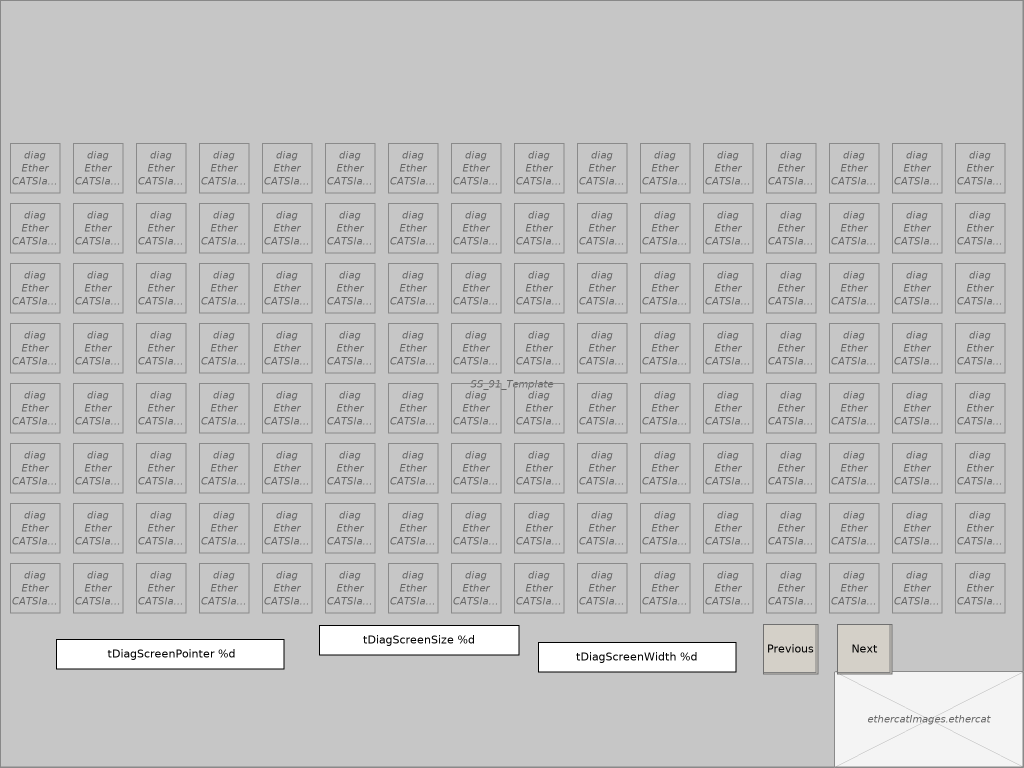
VISUALIZATION DI_02_EtherCAT  // 1024x768
    Frame (0,0 1024x768)
        shows SS_91_Template(header := HMIData.hmiHeader)
    Frame (10,143 50x50)
        shows diagEtherCATSlave(dataValues := etherCATdiag.diagScreen[1])
    Frame (73,143 50x50)
        shows diagEtherCATSlave(dataValues := etherCATdiag.diagScreen[2])
    Frame (136,143 50x50)
        shows diagEtherCATSlave(dataValues := etherCATdiag.diagScreen[3])
    Frame (199,143 50x50)
        shows diagEtherCATSlave(dataValues := etherCATdiag.diagScreen[4])
    Frame (262,143 50x50)
        shows diagEtherCATSlave(dataValues := etherCATdiag.diagScreen[5])
    Frame (325,143 50x50)
        shows diagEtherCATSlave(dataValues := etherCATdiag.diagScreen[6])
    Frame (388,143 50x50)
        shows diagEtherCATSlave(dataValues := etherCATdiag.diagScreen[7])
    Frame (451,143 50x50)
        shows diagEtherCATSlave(dataValues := etherCATdiag.diagScreen[8])
    Frame (514,143 50x50)
        shows diagEtherCATSlave(dataValues := etherCATdiag.diagScreen[9])
    Frame (577,143 50x50)
        shows diagEtherCATSlave(dataValues := etherCATdiag.diagScreen[10])
    Frame (640,143 50x50)
        shows diagEtherCATSlave(dataValues := etherCATdiag.diagScreen[11])
    Frame (703,143 50x50)
        shows diagEtherCATSlave(dataValues := etherCATdiag.diagScreen[12])
    Frame (766,143 50x50)
        shows diagEtherCATSlave(dataValues := etherCATdiag.diagScreen[13])
    Frame (829,143 50x50)
        shows diagEtherCATSlave(dataValues := etherCATdiag.diagScreen[14])
    Frame (892,143 50x50)
        shows diagEtherCATSlave(dataValues := etherCATdiag.diagScreen[15])
    Frame (955,143 50x50)
        shows diagEtherCATSlave(dataValues := etherCATdiag.diagScreen[16])
    Image (834,671 190x96), image: ethercatImages.ethercat
    Frame (10,203 50x50)
        shows diagEtherCATSlave(dataValues := etherCATdiag.diagScreen[17])
    Frame (73,203 50x50)
        shows diagEtherCATSlave(dataValues := etherCATdiag.diagScreen[18])
    Frame (136,203 50x50)
        shows diagEtherCATSlave(dataValues := etherCATdiag.diagScreen[19])
    Frame (199,203 50x50)
        shows diagEtherCATSlave(dataValues := etherCATdiag.diagScreen[20])
    Frame (262,203 50x50)
        shows diagEtherCATSlave(dataValues := etherCATdiag.diagScreen[21])
    Frame (325,203 50x50)
        shows diagEtherCATSlave(dataValues := etherCATdiag.diagScreen[22])
    Frame (388,203 50x50)
        shows diagEtherCATSlave(dataValues := etherCATdiag.diagScreen[23])
    Frame (451,203 50x50)
        shows diagEtherCATSlave(dataValues := etherCATdiag.diagScreen[24])
    Frame (514,203 50x50)
        shows diagEtherCATSlave(dataValues := etherCATdiag.diagScreen[25])
    Frame (577,203 50x50)
        shows diagEtherCATSlave(dataValues := etherCATdiag.diagScreen[26])
    Frame (640,203 50x50)
        shows diagEtherCATSlave(dataValues := etherCATdiag.diagScreen[27])
    Frame (703,203 50x50)
        shows diagEtherCATSlave(dataValues := etherCATdiag.diagScreen[28])
    Frame (766,203 50x50)
        shows diagEtherCATSlave(dataValues := etherCATdiag.diagScreen[29])
    Frame (829,203 50x50)
        shows diagEtherCATSlave(dataValues := etherCATdiag.diagScreen[30])
    Frame (892,203 50x50)
        shows diagEtherCATSlave(dataValues := etherCATdiag.diagScreen[31])
    Frame (955,203 50x50)
        shows diagEtherCATSlave(dataValues := etherCATdiag.diagScreen[32])
    Frame (10,263 50x50)
        shows diagEtherCATSlave(dataValues := etherCATdiag.diagScreen[33])
    Frame (73,263 50x50)
        shows diagEtherCATSlave(dataValues := etherCATdiag.diagScreen[34])
    Frame (136,263 50x50)
        shows diagEtherCATSlave(dataValues := etherCATdiag.diagScreen[35])
    Frame (199,263 50x50)
        shows diagEtherCATSlave(dataValues := etherCATdiag.diagScreen[36])
    Frame (262,263 50x50)
        shows diagEtherCATSlave(dataValues := etherCATdiag.diagScreen[37])
    Frame (325,263 50x50)
        shows diagEtherCATSlave(dataValues := etherCATdiag.diagScreen[38])
    Frame (388,263 50x50)
        shows diagEtherCATSlave(dataValues := etherCATdiag.diagScreen[39])
    Frame (451,263 50x50)
        shows diagEtherCATSlave(dataValues := etherCATdiag.diagScreen[40])
    Frame (514,263 50x50)
        shows diagEtherCATSlave(dataValues := etherCATdiag.diagScreen[41])
    Frame (577,263 50x50)
        shows diagEtherCATSlave(dataValues := etherCATdiag.diagScreen[42])
    Frame (640,263 50x50)
        shows diagEtherCATSlave(dataValues := etherCATdiag.diagScreen[43])
    Frame (703,263 50x50)
        shows diagEtherCATSlave(dataValues := etherCATdiag.diagScreen[44])
    Frame (766,263 50x50)
        shows diagEtherCATSlave(dataValues := etherCATdiag.diagScreen[45])
    Frame (829,263 50x50)
        shows diagEtherCATSlave(dataValues := etherCATdiag.diagScreen[46])
    Frame (892,263 50x50)
        shows diagEtherCATSlave(dataValues := etherCATdiag.diagScreen[47])
    Frame (955,263 50x50)
        shows diagEtherCATSlave(dataValues := etherCATdiag.diagScreen[48])
    Frame (10,323 50x50)
        shows diagEtherCATSlave(dataValues := etherCATdiag.diagScreen[49])
    Frame (73,323 50x50)
        shows diagEtherCATSlave(dataValues := etherCATdiag.diagScreen[50])
    Frame (136,323 50x50)
        shows diagEtherCATSlave(dataValues := etherCATdiag.diagScreen[51])
    Frame (199,323 50x50)
        shows diagEtherCATSlave(dataValues := etherCATdiag.diagScreen[52])
    Frame (262,323 50x50)
        shows diagEtherCATSlave(dataValues := etherCATdiag.diagScreen[53])
    Frame (325,323 50x50)
        shows diagEtherCATSlave(dataValues := etherCATdiag.diagScreen[54])
    Frame (388,323 50x50)
        shows diagEtherCATSlave(dataValues := etherCATdiag.diagScreen[55])
    Frame (451,323 50x50)
        shows diagEtherCATSlave(dataValues := etherCATdiag.diagScreen[56])
    Frame (514,323 50x50)
        shows diagEtherCATSlave(dataValues := etherCATdiag.diagScreen[57])
    Frame (577,323 50x50)
        shows diagEtherCATSlave(dataValues := etherCATdiag.diagScreen[58])
    Frame (640,323 50x50)
        shows diagEtherCATSlave(dataValues := etherCATdiag.diagScreen[59])
    Frame (703,323 50x50)
        shows diagEtherCATSlave(dataValues := etherCATdiag.diagScreen[60])
    Frame (766,323 50x50)
        shows diagEtherCATSlave(dataValues := etherCATdiag.diagScreen[61])
    Frame (829,323 50x50)
        shows diagEtherCATSlave(dataValues := etherCATdiag.diagScreen[62])
    Frame (892,323 50x50)
        shows diagEtherCATSlave(dataValues := etherCATdiag.diagScreen[63])
    Frame (955,323 50x50)
        shows diagEtherCATSlave(dataValues := etherCATdiag.diagScreen[64])
    Frame (10,383 50x50)
        shows diagEtherCATSlave(dataValues := etherCATdiag.diagScreen[65])
    Frame (73,383 50x50)
        shows diagEtherCATSlave(dataValues := etherCATdiag.diagScreen[66])
    Frame (136,383 50x50)
        shows diagEtherCATSlave(dataValues := etherCATdiag.diagScreen[67])
    Frame (199,383 50x50)
        shows diagEtherCATSlave(dataValues := etherCATdiag.diagScreen[68])
    Frame (262,383 50x50)
        shows diagEtherCATSlave(dataValues := etherCATdiag.diagScreen[69])
    Frame (325,383 50x50)
        shows diagEtherCATSlave(dataValues := etherCATdiag.diagScreen[70])
    Frame (388,383 50x50)
        shows diagEtherCATSlave(dataValues := etherCATdiag.diagScreen[71])
    Frame (451,383 50x50)
        shows diagEtherCATSlave(dataValues := etherCATdiag.diagScreen[72])
    Frame (514,383 50x50)
        shows diagEtherCATSlave(dataValues := etherCATdiag.diagScreen[73])
    Frame (577,383 50x50)
        shows diagEtherCATSlave(dataValues := etherCATdiag.diagScreen[74])
    Frame (640,383 50x50)
        shows diagEtherCATSlave(dataValues := etherCATdiag.diagScreen[75])
    Frame (703,383 50x50)
        shows diagEtherCATSlave(dataValues := etherCATdiag.diagScreen[76])
    Frame (766,383 50x50)
        shows diagEtherCATSlave(dataValues := etherCATdiag.diagScreen[77])
    Frame (829,383 50x50)
        shows diagEtherCATSlave(dataValues := etherCATdiag.diagScreen[78])
    Frame (892,383 50x50)
        shows diagEtherCATSlave(dataValues := etherCATdiag.diagScreen[79])
    Frame (955,383 50x50)
        shows diagEtherCATSlave(dataValues := etherCATdiag.diagScreen[80])
    Frame (10,443 50x50)
        shows diagEtherCATSlave(dataValues := etherCATdiag.diagScreen[81])
    Frame (73,443 50x50)
        shows diagEtherCATSlave(dataValues := etherCATdiag.diagScreen[82])
    Frame (136,443 50x50)
        shows diagEtherCATSlave(dataValues := etherCATdiag.diagScreen[83])
    Frame (199,443 50x50)
        shows diagEtherCATSlave(dataValues := etherCATdiag.diagScreen[84])
    Frame (262,443 50x50)
        shows diagEtherCATSlave(dataValues := etherCATdiag.diagScreen[85])
    Frame (325,443 50x50)
        shows diagEtherCATSlave(dataValues := etherCATdiag.diagScreen[86])
    Frame (388,443 50x50)
        shows diagEtherCATSlave(dataValues := etherCATdiag.diagScreen[87])
    Frame (451,443 50x50)
        shows diagEtherCATSlave(dataValues := etherCATdiag.diagScreen[88])
    Frame (514,443 50x50)
        shows diagEtherCATSlave(dataValues := etherCATdiag.diagScreen[89])
    Frame (577,443 50x50)
        shows diagEtherCATSlave(dataValues := etherCATdiag.diagScreen[90])
    Frame (640,443 50x50)
        shows diagEtherCATSlave(dataValues := etherCATdiag.diagScreen[91])
    Frame (703,443 50x50)
        shows diagEtherCATSlave(dataValues := etherCATdiag.diagScreen[92])
    Frame (766,443 50x50)
        shows diagEtherCATSlave(dataValues := etherCATdiag.diagScreen[93])
    Frame (829,443 50x50)
        shows diagEtherCATSlave(dataValues := etherCATdiag.diagScreen[94])
    Frame (892,443 50x50)
        shows diagEtherCATSlave(dataValues := etherCATdiag.diagScreen[95])
    Frame (955,443 50x50)
        shows diagEtherCATSlave(dataValues := etherCATdiag.diagScreen[96])
    Frame (10,503 50x50)
        shows diagEtherCATSlave(dataValues := etherCATdiag.diagScreen[97])
    Frame (73,503 50x50)
        shows diagEtherCATSlave(dataValues := etherCATdiag.diagScreen[98])
    Frame (136,503 50x50)
        shows diagEtherCATSlave(dataValues := etherCATdiag.diagScreen[99])
    Frame (199,503 50x50)
        shows diagEtherCATSlave(dataValues := etherCATdiag.diagScreen[100])
    Frame (262,503 50x50)
        shows diagEtherCATSlave(dataValues := etherCATdiag.diagScreen[101])
    Frame (325,503 50x50)
        shows diagEtherCATSlave(dataValues := etherCATdiag.diagScreen[102])
    Frame (388,503 50x50)
        shows diagEtherCATSlave(dataValues := etherCATdiag.diagScreen[103])
    Frame (451,503 50x50)
        shows diagEtherCATSlave(dataValues := etherCATdiag.diagScreen[104])
    Frame (514,503 50x50)
        shows diagEtherCATSlave(dataValues := etherCATdiag.diagScreen[105])
    Frame (577,503 50x50)
        shows diagEtherCATSlave(dataValues := etherCATdiag.diagScreen[106])
    Frame (640,503 50x50)
        shows diagEtherCATSlave(dataValues := etherCATdiag.diagScreen[107])
    Frame (703,503 50x50)
        shows diagEtherCATSlave(dataValues := etherCATdiag.diagScreen[108])
    Frame (766,503 50x50)
        shows diagEtherCATSlave(dataValues := etherCATdiag.diagScreen[109])
    Frame (829,503 50x50)
        shows diagEtherCATSlave(dataValues := etherCATdiag.diagScreen[110])
    Frame (892,503 50x50)
        shows diagEtherCATSlave(dataValues := etherCATdiag.diagScreen[111])
    Frame (955,503 50x50)
        shows diagEtherCATSlave(dataValues := etherCATdiag.diagScreen[112])
    Frame (10,563 50x50)
        shows diagEtherCATSlave(dataValues := etherCATdiag.diagScreen[113])
    Frame (73,563 50x50)
        shows diagEtherCATSlave(dataValues := etherCATdiag.diagScreen[114])
    Frame (136,563 50x50)
        shows diagEtherCATSlave(dataValues := etherCATdiag.diagScreen[115])
    Frame (199,563 50x50)
        shows diagEtherCATSlave(dataValues := etherCATdiag.diagScreen[116])
    Frame (262,563 50x50)
        shows diagEtherCATSlave(dataValues := etherCATdiag.diagScreen[117])
    Frame (325,563 50x50)
        shows diagEtherCATSlave(dataValues := etherCATdiag.diagScreen[118])
    Frame (388,563 50x50)
        shows diagEtherCATSlave(dataValues := etherCATdiag.diagScreen[119])
    Frame (451,563 50x50)
        shows diagEtherCATSlave(dataValues := etherCATdiag.diagScreen[120])
    Frame (514,563 50x50)
        shows diagEtherCATSlave(dataValues := etherCATdiag.diagScreen[121])
    Frame (577,563 50x50)
        shows diagEtherCATSlave(dataValues := etherCATdiag.diagScreen[122])
    Frame (640,563 50x50)
        shows diagEtherCATSlave(dataValues := etherCATdiag.diagScreen[123])
    Frame (703,563 50x50)
        shows diagEtherCATSlave(dataValues := etherCATdiag.diagScreen[124])
    Frame (766,563 50x50)
        shows diagEtherCATSlave(dataValues := etherCATdiag.diagScreen[125])
    Frame (829,563 50x50)
        shows diagEtherCATSlave(dataValues := etherCATdiag.diagScreen[126])
    Frame (892,563 50x50)
        shows diagEtherCATSlave(dataValues := etherCATdiag.diagScreen[127])
    Frame (955,563 50x50)
        shows diagEtherCATSlave(dataValues := etherCATdiag.diagScreen[128])
    Button (763,624 55x50), "Previous"
        tap etherCATdiag.btnPrevious
    Button (837,624 55x50), "Next"
        tap etherCATdiag.btnNext
    Rectangle (56,639 228x30), "tDiagScreenPointer %d", text variable: pouEtherCATdiag.tDiagScreenPointer
    Rectangle (319,625 200x30), "tDiagScreenSize %d", text variable: pouEtherCATdiag.tDiagScreenSize
    Rectangle (538,642 198x30), "tDiagScreenWidth %d", text variable: pouEtherCATdiag.tDiagScreenWidth
END_VISUALIZATION

(* stored: Version 1.1.0.1, ProductVersion 3.1.4024.12
   Visu DI_02_EtherCAT: Id {14ac5115-3a58-4a05-8fe9-a2630b3c459e} *)
